Staubli VAL3: clkAllOff.pgx

program clkAllOff()
  local num index
begin
  for index=0 to 31
    if statusValves[index]==1
      call toggleValve(index)
    endIf
  endFor
end
